FUNCTION_BLOCK my_sensor (* Basic Function Block Type *)
  (* Standard: 61499-2 *)
  (* Version 0.2, 2003-12-04, JHC, Rockwell Automation, Renamed for better indexing. *)
  (* Version 0.1, 2002-11-05, JHC, Rockwell Automation, Corrected missing ST element in Algorithm REQ. *)
  (* Version 0.0, 2000-05-30, JHC, Rockwell Automation *)
  (* Compiler header: package fb.rt.pnp; *)
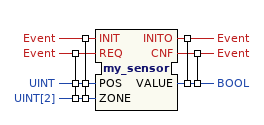
  EVENT_INPUT
    INIT WITH POS, ZONE; (* Initialization Request *)
    REQ WITH POS, ZONE; (* Normal Execution Request *)
  END_EVENT
  EVENT_OUTPUT
    INITO WITH VALUE; (* Initialization Confirm *)
    CNF WITH VALUE; (* Execution Confirmation *)
  END_EVENT
  VAR_INPUT
    POS : UINT; (* Input event qualifier *)
    ZONE : ARRAY [0..1] OF UINT;
  END_VAR
  VAR_OUTPUT
    VALUE : BOOL; (* Output event qualifier *)
  END_VAR
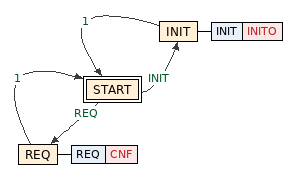
  EC_STATES
    START; (* Initial State *)
    INIT : INIT -> INITO; (* Initialization *)
    REQ : REQ -> CNF; (* Normal execution *)
  END_STATES
  EC_TRANSITIONS
    START TO INIT := INIT;
    INIT TO START := 1;
    START TO REQ := REQ;
    REQ TO START := 1;
  END_TRANSITIONS
  ALGORITHM INIT IN ST: (* Initialization algorithm *)
VALUE:=FALSE;
  END_ALGORITHM
  ALGORITHM REQ IN Java: (* Normally executed algorithm *)
if((POS.value>=((UINT)ZONE.value[0]).value)&(POS.value<=((UINT)ZONE.value[1]).value)){
VALUE.value=true;
//System.out.println("Sensor True " + POS.value);
}
else{
VALUE.value=false;
}
  END_ALGORITHM
END_FUNCTION_BLOCK
